{attribute 'qualified_only'}
VAR_GLOBAL
	adsMajorNetwork : AdsTcpUnitEx;
END_VAR

(* stored: Version 1.1.0.1, ProductVersion 3.1.4024.11
   GVL COM: Id {23b5e941-7a30-44ab-b048-0bb85aca0ea5} *)
